// TIA Portal V20 export
DATA_BLOCK "DB_UDI"   // DB37
// stored: MemoryReserve 100, Namespace LineC1
   VAR
      LineC1 : Struct
         Upstream : Struct
            Conveyor : Array[_.minC1.._.maxC1] of Bool;
         END_STRUCT;
         DownstreamAccu : Struct
            Conveyor : Array[_.minC1.._.maxC1] of Bool;
         END_STRUCT;
         Interlock : Struct
            Conveyor : Array[_.minC1.._.maxC1] of Bool;
         END_STRUCT;
         Fault : Struct
            Conveyor : Array[_.minC1.._.maxC1] of Bool;
         END_STRUCT;
         Merging1 : Struct
            "Timer" : Struct
               StraightTote : TON_TIME;
               ArmTote { S7_SetPoint := 'True'} : TON_TIME;
            END_STRUCT;
            Priority : Struct
               Straight : Bool;
               Arm : Bool;
            END_STRUCT;
         END_STRUCT;
         Merging2 : Struct
            "Timer" : Struct
               StraightTote : TON_TIME;
               ArmTote { S7_SetPoint := 'True'} : TON_TIME;
            END_STRUCT;
            Priority : Struct
               Straight : Bool;
               Arm : Bool;
            END_STRUCT;
         END_STRUCT;
      END_STRUCT;
   END_VAR
BEGIN
END_DATA_BLOCK
